# B&R Automation Studio project Tmp_Recorder_V1
Automation Studio 4.5.5.113 SP; technology packages: mapp 5.8.1, mappView 5.8.1

## Configuration X20CPU

CPU X20CP1583, AutomationRuntime B4.53, Build 4.1.2, Vc V4.52.0

CPU X20CP3687X, AutomationRuntime C4.90, Build 4.1.2, Vc V4.52.0

### Task classes (Cpu.sw)
```
Cyclic#8:
  Recorder_1 <- mappRecorder.Recorder_1.prg
Binaries: udbdef, mvLoader, TCData, arsvcreg, Config, sysconf, ashwd, ashwac, asfw, iomap, Role, User, arconfig, OpcUaMap
Libraries: FileIO, runtime, AsBrStr, standard, AsBrWStr, MpBase, sys_lib, IecCheck, asieccon, AsIODiag, MpData, DataObj, brsystem, astime, MpServer, MpFile, AsHttp, AsMem
```

### Task classes (Cpu.sw)
```
Cyclic#4:
  YourTask <- mappRecorder.YourTask.prg
Cyclic#8:
  Recorder_1 <- mappRecorder.Recorder_1.prg
Binaries: udbdef, mvLoader, TCData, arsvcreg, Config, sysconf, ashwd, ashwac, asfw, iomap, Role, User, arconfig, OpcUaMap
Libraries: FileIO, runtime, AsBrStr, standard, AsBrWStr, MpBase, sys_lib, IecCheck, asieccon, AsIODiag, MpData, DataObj, brsystem, astime, MpServer, MpFile, AsHttp, AsMem, MpCom
```

### Hardware
```
X20CP3687X : X20CP3687X v1.7.2.0
  Connector IF2:
    ActivateDevice = 1
  Connector IF3:
    DNAConfiguration = manual
    CycleTime = 2000
  ConfigurationID = Tmp_Recorder
  UserPartitionSize = 200
  AutomaticTransferOfUserfiles = on
  VolatileGlobalPvSize = 300000
  Cyclic8Stack = 20000
  FileDevice1
  FileDeviceName1 = RECORDER_DEVICE
  FileDevicePath1 = F:/
  FileDevice2
  FileDeviceName2 = SIM_DEVICE
  FileDevicePath2 = C:/Temp
  FtpUser1
  FtpUsername1 = br
  FtpUserPassword1 = B+jJgvp9Np1Nx73dPwFagqyDiJQWzomgOnJThoU8F9Q=  // password
  FtpUserSalt1 = Snq9ellj
  FTPAccessRight1 = 0
  ActivateSdm = 0
  ActivateOpcUa = 1
  OpcUaInformationModels_PV_Version = 1
```

### Config_1.mpdatarecorder - X20CP1583/mappServices/Config_1.mpdatarecorder
```
Element gDataRecorder_1 (Type=mpdatarecorder)
```

- Physical/X20CPU/X20CP3687X/mappServices/Config_1.mpdatarecorder: same as Physical/X20CPU/X20CP1583/mappServices/Config_1.mpdatarecorder
## Logical view

Binary libraries used (declarations not repeated): operator, runtime, astime, AsIecCon, FileIO, AsBrStr, AsBrWStr, standard, sys_lib, IecCheck, AsIODiag, DataObj, brsystem, AsHttp, AsMem, MpFile 5.15.0, MpBase 5.15.0, MpCom 5.15.0, MpData 5.15.0, MpServer 5.15.0

### Package Logical/Libraries - Global libraries

- Visualisation Logical/mappView (not shown)

### DatTypes.typ
```iecst
(*------------------------------------------------------------------------------------------------------------------------------------------------------------------------------------------------------------------------*)
(*Global enumerations*)

TYPE
	datSTATE :
		( (*Recorder managment state machine*)
		DAT_WAIT,
		DAT_REG_VAR,
		DAT_READ_DIR,
		DAT_READ_DIR_1,
		DAT_READ_DIR_2,
		DAT_READ_DIR_3,
		DAT_CFG_READ,
		DAT_CFG_WRITE,
		DAT_RECORD,
		DAT_DELETE,
		DAT_VIEW,
		DAT_DOWNLOAD,
		DAT_DOWNLOAD_1,
		DAT_DOWNLOAD_2,
		DAT_DOWNLOAD_3,
		DAT_DOWNLOAD_4,
		DAT_LOAD_VARS,
		DAT_LOAD_VARS_1,
		DAT_LOAD_VARS_2,
		DAT_LOAD_VARS_3,
		DAT_ERROR
		);
END_TYPE

(*------------------------------------------------------------------------------------------------------------------------------------------------------------------------------------------------------------------------*)
(*Global structure*)

TYPE
	datERR : 	STRUCT  (*Recorder managment error structure*)
		Text : WSTRING[200]; (* Error text *)
		State : datSTATE; (* Error step *)
	END_STRUCT;
	datCMD : 	STRUCT  (*Recorder managment command structure*)
		Init : BOOL := TRUE; (*Initialize recorder structure*)
		Record : BOOL; (*Enable recording*)
		Trigger : BOOL; (*Trigger recording*)
		Delete : BOOL; (*Delete selected file *)
		View : BOOL; (*View selected file*)
		Download : BOOL; (*Download selected file*)
		LoadConfig : BOOL; (*Load variable configuration from file*)
		ErrorReset : BOOL; (*Reset pending errors*)
	END_STRUCT;
	datPAR : 	STRUCT  (*Recorder managment parameter structure*)
		RecordName : STRING[DAT_NAME_LENGTH]; (*Record name for command delete and view*)
		RecordNameNew : STRING[DAT_NAME_LENGTH]; (*Record name for command record*)
		RecordMode : MpDataRecordModeEnum; (*Recording mode*)
		RecordInterval : TIME := T#2000ms;
		IsRecording : BOOL; (*Indicates that recording is active*)
		SamplesNum : UDINT; (*Number of recorded samples*)
		Initialized : BOOL; (*Indicates that recorder managment was initialized*)
		VisuSlotID : USINT; (*ID for connected web connection*)
	END_STRUCT;
	datDAT : 	STRUCT  (*Recorder managment data structure*)
		RecordNames : ARRAY[0..DAT_MAX_NUM]OF STRING[DAT_NAME_LENGTH]; (*Recorder unicode name*)
		RecordNum : UINT; (*Number of recorded files*)
	END_STRUCT;
	datVIS : 	STRUCT  (*Recorder managment visualization structure*)
		RecordNames : ARRAY[0..DAT_MAX_NUM]OF STRING[DAT_VIS_LENGTH]; (*Recorder file size*)
		RecordNum : UINT; (*Number of records*)
		RecordFilter : STRING[DAT_NAME_LENGTH]; (*Filter for record names*)
		RecordSelected : STRING[DAT_VIS_LENGTH]; (*Selected record for command delete or view*)
		RecordDoubleClick : USINT; (*TrackDoubleClick event*)
		EnableButtons : BOOL;
		ViewFilePath : STRING[DAT_VIS_LENGTH]; (*Full path for viewing file*)
		ViewFile : BOOL; (*Show message box on error*)
		DownloadFileUrl : STRING[200]; (*File upload and download url*)
		ShowMessageBoxError : BOOL; (*Show message box on error*)
	END_STRUCT;
	datMAIN : 	STRUCT  (*Recorder managment main structure*)
		CMD : datCMD; (*Command structure *)
		PAR : datPAR; (*Parameter structure *)
		DAT : datDAT; (*Data structure*)
		VIS : ARRAY[0..DAT_MAX_CLIENTS_ID]OF datVIS; (*Visualization structure*)
		ERR : datERR; (*Error structure *)
		StatusText : WSTRING[100]; (*Shows the result of the last command*)
		StatusNo : DINT; (*Error number *)
	END_STRUCT;
END_TYPE

(*------------------------------------------------------------------------------------------------------------------------------------------------------------------------------------------------------------------------*)
(*Structure that contains the recorder variables*)

TYPE
	datVariable : 	STRUCT
		Temperature1 : INT := 11;
		Temperature2 : INT := 22;
		MotorSpeed : DINT := 33;
		Position : REAL := 44.55;
	END_STRUCT;
END_TYPE
```

### DatVariables.var
```iecst
(*------------------------------------------------------------------------------------------------------------------------------------------------------------------------------------------------------------------------*)
(*Configuration for recorder managment*)
VAR CONSTANT
	DAT_MAX_NUM : USINT := 100; (*Maximum number of record files*)
	DAT_NAME_LENGTH : USINT := 40; (*Maximum length for a record name*)
	DAT_VIS_LENGTH : USINT := 120; (*Make this DAT_NAME_LENGTH  x3*)
	DAT_MAX_CLIENTS_ID : USINT := 2; (*Highest client ID for concurrent web client connections. Do not change this number.*)
END_VAR
VAR
	DAT_VIEW_FILTER : ARRAY[0..9] OF STRING[5] := ['csv','pdf',8('')]; (*Files extensions than can be used with the view command*)
END_VAR
VAR CONSTANT
	DAT_DOWNLOAD_SIZE : UDINT := 500000; (*Maximum size of memory allocated for uploading and downloading files*)
	DAT_VAR_NUM : USINT := 10; (*Maximum number of variables that can be registered*)
	DAT_THIS_TASK : STRING[40] := 'Recorder_1'; (*Name of this task and the global variables structure*)
	DAT_DEVICE : STRING[80] := 'RECORDER_DEVICE'; (*Device name for the recorder data defined under File Devices in the CPU configuration*)
	DAT_CONFIG : STRING[80] := 'var_list.csv'; (*File with a list of variables in CSV format*)
END_VAR
VAR
	DAT_MPLINK : {REDUND_UNREPLICABLE} STRING[80] := 'gDataRecorder_1'; (*mappRecoreer link name from configuration view*)
END_VAR
(*------------------------------------------------------------------------------------------------------------------------------------------------------------------------------------------------------------------------*)
(*Add you variables to this list*)
VAR
	DAT_VAR_LIST : ARRAY[1..DAT_VAR_NUM] OF STRING[100] := ['YourTask:Temperature1','YourTask:Temperature2','YourTask:MotorSpeed','YourTask:Position',6('')]; (*List of variables to be inlcuded in a record*)
	Recorder_1 : datMAIN; (*Global record structure. The name must match the task name of the recorder managment.*)
END_VAR
```

### Program Logical/mappRecorder/Recorder_1 (IEC)

#### Init.st - Init and local configuration
```iecst
// -------------------------------------------------------------------------------------------------------------------
//	Function:	Data recorder management with mappData
// -------------------------------------------------------------------------------------------------------------------
PROGRAM _INIT
	// ----------------------------------------------------------------------------------------
	// The following settings can be adjusted
	IF(DiagCpuIsSimulated()) THEN
		DeviceName 	:= 'SIM_DEVICE';	// Device name from the CPU configuration for simulation
	ELSE
		DeviceName 	:= DAT_DEVICE;		// Device name from the CPU configuration for X20CPU
	END_IF

	// ----------------------------------------------------------------------------------------
	// Dont change anything below this line
	// ----------------------------------------------------------------------------------------

	// ----------------------------------------------------------------------------------------
	// Make sure global variable structure and task name are correct
	taskStatus := ST_ident(ADR(DAT_THIS_TASK), taskGroup, ADR(taskID));
	pvStatus := PV_xgetadr(ADR(DAT_THIS_TASK), ADR(pvADR), ADR(pvLEN));
	// Connect global and local structure
	IF(pvStatus = 0) THEN
		RECORDER ACCESS pvADR;
		brsmemset(ADR(RECORDER.ERR), 0 , SIZEOF(RECORDER.ERR));
		RECORDER.PAR.Initialized := FALSE;
	END_IF

	// ----------------------------------------------------------------------------------------
	// Get mapp link information
	MpComGetLink_0.Enable := TRUE;
	MpComGetLink_0.ComponentName := ADR(DAT_MPLINK);
	MpComGetLink_0();
	// Create error
	IF(MpComGetLink_0.Error) THEN
		rec_state := CreateError(ADR(RECORDER), ERR_DAT_MPLINK, "mplink name is incorrect", rec_state);
	END_IF

	// ----------------------------------------------------------------------------------------
	// Allocate memory for file upload and download
	AsMemPartCreate_0.enable	:= TRUE;
	AsMemPartCreate_0.len		:= DAT_DOWNLOAD_SIZE;
	AsMemPartCreate_0();
	IF AsMemPartCreate_0.status <> 0 THEN
		CreateError(ADR(RECORDER), ERR_MEM_ALLOC, "file upload and download alloc failed", rec_state);
	ELSE
		AsMemPartAllocClear_0.enable	:= TRUE;
		AsMemPartAllocClear_0.ident		:= AsMemPartCreate_0.ident;
		AsMemPartAllocClear_0.len		:= DAT_DOWNLOAD_SIZE;
		AsMemPartAllocClear_0();
		IF AsMemPartCreate_0.status <> 0 THEN
			CreateError(ADR(RECORDER), ERR_MEM_ALLOC, "file upload and download clear failed", rec_state);
		END_IF
	END_IF
END_PROGRAM
```

#### Main.st - Cyclic code
```iecst
// -------------------------------------------------------------------------------------------------------------------
//	Cylic task for data recorder management
// -------------------------------------------------------------------------------------------------------------------
PROGRAM _CYCLIC
	// --------------------------------------------------------------------------------------------------------------------
	// Make sure task name and global structure correct
	IF(pvStatus <> 0) THEN
		RETURN;
	END_IF
	IF(taskStatus <> 0) THEN
		rec_state := CreateError(ADR(RECORDER), ERR_DAT_TASK_NAME, "Task name is incorrect", rec_state);
		RETURN;
	END_IF

	// --------------------------------------------------------------------------------------------------------------------
	// Make sure we dont exceed maximum number of web clients
	IF(RECORDER.PAR.VisuSlotID > DAT_MAX_CLIENTS_ID) THEN
		rec_state := CreateError(ADR(RECORDER), ERR_DAT_TOO_MANY_CLIENTS, "More than 3 clients try to connect to data recorder", rec_state);
		RETURN;
	END_IF

	// --------------------------------------------------------------------------------------------------------------------
	// Cyclic function calls
	MpDataRecorder_0();
	RECORDER.PAR.IsRecording := MpDataRecorder_0.Recording;
	RECORDER.PAR.SamplesNum := MpDataRecorder_0.Info.TotalSamples;
	MpDataRecorder_0.RecordMode := RECORDER.PAR.RecordMode;
	MpDataRecorder_0.SamplingTime := RECORDER.PAR.RecordInterval;

		// -------------------------------------------------------------------------------------------------------------------
	// Recorder managment state machine
		// -------------------------------------------------------------------------------------------------------------------
	CASE rec_state OF
		// --------------------------------------------------------------------------------------------------------------------
		// Wait for command
		// --------------------------------------------------------------------------------------------------------------------
		DAT_WAIT:
			// Set OK state
			RECORDER.StatusNo := ERR_OK;
			// --------------------------------------------------------------------------------------------------------------------
			// Track filter change and data refresh
			IF ((brwcscmp(ADR(RecordFilterOld[VisuSlotID]), ADR(RECORDER.VIS[VisuSlotID].RecordFilter)) <> 0) OR (RecordNumOld[VisuSlotID] <> RECORDER.DAT.RecordNum)) THEN
				brsmemset(ADR(RECORDER.VIS[VisuSlotID].RecordNames), 0, SIZEOF(RECORDER.VIS[VisuSlotID].RecordNames));
				idy := 0;
				IF(RECORDER.DAT.RecordNum > 0) THEN
					FOR idx:=0 TO RECORDER.DAT.RecordNum - 1 DO
						// --------------------------------------------------------------------------------
						// Verify that file name contains filter
						IF (brsstrlen(ADR(RECORDER.VIS[VisuSlotID].RecordFilter)) = 0 OR IsInstr(ADR(RECORDER.DAT.RecordNames[idx]), ADR(RECORDER.VIS[VisuSlotID].RecordFilter))) > 0 THEN
							String2DataProvider(ADR(RECORDER.DAT.RecordNames[idx]), ADR(tmpStr1));
							RECORDER.VIS[VisuSlotID].RecordNames[idy] := tmpStr1;
							idy := idy + 1;
						END_IF
					END_FOR;
					brsstrcpy(ADR(RecordFilterOld[VisuSlotID]), ADR(RECORDER.VIS[VisuSlotID].RecordFilter));
				END_IF
				RecordNumOld[VisuSlotID] := RECORDER.DAT.RecordNum;
				RECORDER.VIS[VisuSlotID].RecordNum := idy;
				// Enable/Disable delete button
				IF(RECORDER.VIS[VisuSlotID].RecordNum > 0) THEN
					RECORDER.VIS[VisuSlotID].EnableButtons := TRUE;
				ELSE
					RECORDER.VIS[VisuSlotID].EnableButtons := FALSE;
				END_IF
			END_IF

			// ------------------------------------------------------------------------------------------------
			// Handle double click for file open
			IF(RECORDER.VIS[VisuSlotID].RecordDoubleClick > 0) THEN
				DoubleClickRecordName[VisuSlotID].PT := 50;
				DoubleClickRecordName[VisuSlotID].IN := 1;
				DoubleClickRecordName[VisuSlotID]();
				// Open selected file
				IF(RECORDER.VIS[VisuSlotID].RecordDoubleClick > 1) THEN
					DoubleClickRecordName[VisuSlotID].IN := 0;
					DoubleClickRecordName[VisuSlotID]();
					RECORDER.VIS[VisuSlotID].RecordDoubleClick := 0;
					RECORDER.PAR.VisuSlotID := VisuSlotID;
					RECORDER.CMD.View := TRUE;
				END_IF
			END_IF
			IF(DoubleClickRecordName[VisuSlotID].Q) THEN
				DoubleClickRecordName[VisuSlotID].IN := 0;
				DoubleClickRecordName[VisuSlotID]();
				IF(RECORDER.VIS[VisuSlotID].RecordDoubleClick > 0) THEN
					RECORDER.VIS[VisuSlotID].RecordDoubleClick := RECORDER.VIS[VisuSlotID].RecordDoubleClick - 1;
				END_IF
			END_IF

			// Cylce through the client web seesions
			VisuSlotID := VisuSlotID + 1;
			IF(VisuSlotID > DAT_MAX_CLIENTS_ID) THEN
				VisuSlotID := 0;
			END_IF

			// ----------------------------------------------------------------------------------------
			// Command refresh
			IF (RECORDER.CMD.Init = TRUE) THEN
				// Reset data structure and trigger name refresh for vis
				brsmemset(ADR(RECORDER.DAT), 0, SIZEOF(RECORDER.DAT));
				brsmemset(ADR(RecordNumOld), 16#FF, SIZEOF(RecordNumOld));
				pvCnt := 1;
				rec_state := DAT_CFG_READ;
			// ----------------------------------------------------------------------------------------
			// Command continues recording
			ELSIF (RECORDER.CMD.Record = TRUE) THEN
				tmpWStr1 := "continues recording...";
				rec_state := DAT_CFG_WRITE;
			// ----------------------------------------------------------------------------------------
			// Command trigger recording
			ELSIF (RECORDER.CMD.Trigger = TRUE) THEN
				tmpWStr1 := "recording by trigger...";
				rec_state := DAT_RECORD;
			// ----------------------------------------------------------------------------------------
			// Command delete recording
			ELSIF (RECORDER.CMD.Delete = TRUE AND RECORDER.PAR.RecordName <> '') THEN
				animation := WorkingStatus(ADR(RECORDER), ADR("deleting recording..."), animation);
				RecordName := RECORDER.PAR.RecordName;
				rec_state := DAT_DELETE;
			// ----------------------------------------------------------------------------------------
			// Command view file
			ELSIF (RECORDER.CMD.View = TRUE AND RECORDER.VIS[RECORDER.PAR.VisuSlotID].RecordSelected <> '') THEN
				RECORDER.VIS[RECORDER.PAR.VisuSlotID].ViewFilePath := '';
				//RecordName := RECORDER.PAR.RecordName;
				rec_state := DAT_VIEW;
			// ----------------------------------------------------------------------------------------
			// Download selected file
			ELSIF (RECORDER.CMD.Download = 1 AND RECORDER.PAR.RecordName <> '') THEN
				RECORDER.VIS[RECORDER.PAR.VisuSlotID].DownloadFileUrl := '';
				RecordName := RECORDER.PAR.RecordName;
				rec_state := DAT_DOWNLOAD;
			// ----------------------------------------------------------------------------------------
			// Load variable configuration file
			ELSIF (RECORDER.CMD.LoadConfig = 1) THEN
				rec_state := DAT_LOAD_VARS;
			END_IF

			// ----------------------------------------------------------------------------------------
			// Check parameters
			IF (RECORDER.CMD.Init OR RECORDER.CMD.Delete OR RECORDER.CMD.View OR RECORDER.CMD.Download OR RECORDER.CMD.LoadConfig OR RECORDER.CMD.Record) THEN
				// Set busy state
				RECORDER.StatusNo := ERR_FUB_BUSY;
				// Make sure recorder was intialized
				IF (NOT RECORDER.CMD.Init AND (RECORDER.CMD.Delete OR RECORDER.CMD.View) AND NOT RECORDER.PAR.Initialized) THEN
					rec_state := CreateError(ADR(RECORDER), ERR_DAT_NOT_INITIALIZED, "recorder is not initialized", rec_state);
				END_IF
				// Make sure device name is valid
				IF(DeviceName = '') THEN
					rec_state := CreateError(ADR(RECORDER), ERR_DAT_DEV_NAME_EMPTY, "device name is empty", rec_state);
				END_IF
				// Make sure record name is valid
				IF(RECORDER.PAR.RecordName = '' AND (RECORDER.CMD.Delete OR RECORDER.CMD.Download)) THEN
					rec_state := CreateError(ADR(RECORDER), ERR_DAT_NAME_EMPTY, "record name is empty", rec_state);
				END_IF
				// Make sure record name is valid
				IF(RECORDER.PAR.RecordNameNew = '' AND RECORDER.CMD.Record) THEN
					rec_state := CreateError(ADR(RECORDER), ERR_DAT_NAME_EMPTY, "new record name is empty", rec_state);
				END_IF
				// Make sure variable name has at least one entry
				IF(DAT_VAR_LIST[1] = '' AND NOT RECORDER.CMD.LoadConfig) THEN
					rec_state := CreateError(ADR(RECORDER), ERR_DAT_VAR_NAME_EMPTY, "variable name is empty", rec_state);
				END_IF
			END_IF

		// ----------------------------------------------------------------------------------------------------------------------------------
		// Read data configuration
		// ----------------------------------------------------------------------------------------------------------------------------------
		DAT_CFG_READ:
			// Read data configuration
			mappDataCfg.Load := TRUE;

			// ----------------------------------------------------------------------------------------------------------------------------------
			// OK
			IF (mappDataCfg.CommandDone AND NOT mappDataCfg.Error) THEN
				// Reset config function block
				mappDataCfg.Load := FALSE;
				RECORDER.PAR.RecordNameNew := MpDataRecorderCfg.FileNamePattern;
				rec_state := DAT_REG_VAR;
				// ----------------------------------------------------------------------------------------------------------------------------------
				// Error
			ELSIF(mappDataCfg.Error) THEN
				rec_state := CreateError(ADR(RECORDER), mappDataCfg.StatusID, "error reading configuration", rec_state);
			END_IF

		// --------------------------------------------------------------------------------------------------------------------
		// Register variable structure
		// --------------------------------------------------------------------------------------------------------------------
		DAT_REG_VAR:
			MpRecorderRegPar_0[pvCnt].Enable := 1;
			MpRecorderRegPar_0[pvCnt].MpLink := ADR(MpComGetLink_0.MpLink);
			MpRecorderRegPar_0[pvCnt].PVName := ADR(DAT_VAR_LIST[pvCnt]);

			// ----------------------------------------------------------------------------------------
			// OK
			IF (MpRecorderRegPar_0[pvCnt].Active AND NOT MpRecorderRegPar_0[pvCnt].Error) THEN
				pvCnt := pvCnt + 1;
				// Register next variable
				IF((pvCnt >= SIZEOF(DAT_VAR_LIST)/SIZEOF(DAT_VAR_LIST[pvCnt])) OR (DAT_VAR_LIST[pvCnt] = '')) THEN
					rec_state := DAT_READ_DIR;
				END_IF
			// ----------------------------------------------------------------------------------------
			// Error
			ELSIF (MpRecorderRegPar_0[pvCnt].Error) THEN
				tmpWStr1 := "error trying to register variable name ";
				brwcsconv(ADR(tmpWStr2), ADR(DAT_VAR_LIST[pvCnt]), brwU8toUC);
				brwcscat(ADR(tmpWStr1), ADR(tmpWStr2));
				rec_state := CreateError(ADR(RECORDER), MpRecorderRegPar_0[pvCnt].StatusID, tmpWStr1, rec_state);
			END_IF
		// --------------------------------------------------------------------------------------------------------------------
		// Read directory information
		// --------------------------------------------------------------------------------------------------------------------
		DAT_READ_DIR:
			// Show current state
			animation := WorkingStatus(ADR(RECORDER), ADR("reading records..."), animation);
			// ----------------------------------------------------------------------------------------
			// Clear all entrys
			brsmemset(ADR(RECORDER.DAT), 0, SIZEOF(RECORDER.DAT));
			RECORDER.DAT.RecordNum := 0;
			// ----------------------------------------------------------------------------------------
			// Set values and get device dir
			DInfo.enable 	:= 1;
			DInfo.pDevice	:= ADR(DeviceName);
			DInfo();

			// ----------------------------------------------------------------------------------------
			// OK
			IF (DInfo.status = OK) THEN
				rec_state := DAT_READ_DIR_1;
			ELSIF (DInfo.status = fiERR_DEVICE_MANAGER) THEN
				tmpWStr1 := "file device ";
				brwcsconv(ADR(tmpWStr2), ADR(DeviceName), brwU8toUC);
				brwcscat(ADR(tmpWStr1), ADR(tmpWStr2));
				brwcscat(ADR(tmpWStr1), ADR(" is unavailable"));
				rec_state := CreateError(ADR(RECORDER), DInfo.status, tmpWStr1, rec_state);
			// ----------------------------------------------------------------------------------------
			// Error
			ELSIF (DInfo.status <> ERR_FUB_BUSY) THEN
				rec_state := CreateError(ADR(RECORDER), DInfo.status, "error dir info", rec_state);
			END_IF
		// --------------------------------------------------------------------------------------------------------------------
		// Open directory
		// --------------------------------------------------------------------------------------------------------------------
		DAT_READ_DIR_1:
			DOpen.enable 	:= 1;
			DOpen.pDevice	:= ADR(DeviceName);
			DOpen();

			// ----------------------------------------------------------------------------------------
			// OK
			IF (DOpen.status = OK) THEN
				has_oversized_items := FALSE;
				rec_state := DAT_READ_DIR_2;
			// ----------------------------------------------------------------------------------------
			// Error
			ELSIF (DOpen.status <> ERR_FUB_BUSY) THEN
				rec_state := CreateError(ADR(RECORDER), DOpen.status, "error dir open", rec_state);
			END_IF;
		// --------------------------------------------------------------------------------------------------------------------
		// Read file directory information
		// --------------------------------------------------------------------------------------------------------------------
		DAT_READ_DIR_2:
			DRead.enable 	:= 1;
			DRead.ident		:= DOpen.ident;
			DRead.pData 	:= ADR(lDirReadData);
			DRead.data_len 	:= SIZEOF(lDirReadData);
			DRead();

			// ----------------------------------------------------------------------------------------
			// OK
			IF (DRead.status = OK AND lDirReadData.Mode = fiFILE) THEN
				animation := WorkingStatus(ADR(RECORDER), ADR("reading record data..."), animation);
				// Make sure file name does not exceed maximum string size
				IF (brsstrlen(ADR(lDirReadData.Filename)) < DAT_NAME_LENGTH) THEN
					// Copy dir info to string
					brsmemset(ADR(RECORDER.PAR.RecordName), 0, SIZEOF(RECORDER.PAR.RecordName));
					brsstrcpy(ADR(RECORDER.PAR.RecordName), ADR(lDirReadData.Filename));
					// Make sure file extension is CSV or PDF
					IF(brsstrlen(ADR(RECORDER.PAR.RecordName)) > 4 AND ((brsmemcmp(ADR(RECORDER.PAR.RecordName) + (brsstrlen(ADR(RECORDER.PAR.RecordName)) - 4), ADR('.csv'), 4) = 0) OR (brsmemcmp(ADR(RECORDER.PAR.RecordName) + (brsstrlen(ADR(RECORDER.PAR.RecordName)) - 4), ADR('.pdf'), 4) = 0))) THEN
						// ------------------------------------------------------------------------------------
						// Verify that we still have space in list
						IF (RECORDER.DAT.RecordNum <= DAT_MAX_NUM) THEN
							// Generate ASCII data, insert record into list
							InsertRecName(ADR(RECORDER), RECORDER.PAR.RecordName);
							// Error
						ELSE
							rec_state := CreateError(ADR(RECORDER), ERR_DAT_MAX_NUM, "maximum number of records reached", rec_state);
						END_IF
					END_IF
				ELSE
					has_oversized_items := TRUE;
				END_IF
			// ----------------------------------------------------------------------------------------
			// Last entry reached
			ELSIF (DRead.status = fiERR_NO_MORE_ENTRIES) THEN
				rec_state := DAT_READ_DIR_3;
			// ----------------------------------------------------------------------------------------
			// Error
			ELSIF (DRead.status <> ERR_FUB_BUSY AND DRead.status <> OK) THEN
				rec_state := CreateError(ADR(RECORDER), DRead.status, "error record list read", rec_state);
			END_IF
		// --------------------------------------------------------------------------------------------------------------------
		// Close directory information
		// --------------------------------------------------------------------------------------------------------------------
		DAT_READ_DIR_3:
			DClose.enable 	:= 1;
			DClose.ident	:= DOpen.ident;
			DClose();

			// ----------------------------------------------------------------------------------------
			// OK
			IF (DClose.status = OK) THEN
				// Reset command and return to wait state
				RECORDER.StatusText	:= "initializing complete";
				RECORDER.CMD.Init := 0;
				RECORDER.CMD.LoadConfig := 0;
				RECORDER.CMD.Delete := 0;
				RECORDER.PAR.Initialized := TRUE;
				DClose.ident := 0;
				IF(has_oversized_items) THEN
					rec_state := CreateError(ADR(RECORDER), ERR_DAT_NAME_LENGTH, "one or more record names exceeds maximum length", rec_state);
				ELSE
					rec_state := DAT_WAIT;
				END_IF
			// ----------------------------------------------------------------------------------------
			// Error
			ELSIF (DClose.status <> ERR_FUB_BUSY) THEN
				rec_state := CreateError(ADR(RECORDER), DClose.status, "error dir close", rec_state);
			END_IF

		// ----------------------------------------------------------------------------------------------------------------------------------
		// Write data configuration
		// ----------------------------------------------------------------------------------------------------------------------------------
		DAT_CFG_WRITE:
			// Make sure file extension is CSV or PDF
			IF(brsstrlen(ADR(RECORDER.PAR.RecordNameNew)) <= 4 OR ((brsmemcmp(ADR(RECORDER.PAR.RecordNameNew) + (brsstrlen(ADR(RECORDER.PAR.RecordNameNew)) - 4), ADR('.csv'), 4) <> 0) AND (brsmemcmp(ADR(RECORDER.PAR.RecordNameNew) + (brsstrlen(ADR(RECORDER.PAR.RecordNameNew)) - 4), ADR('.pdf'), 4) <> 0))) THEN
				// Make sure record name is not too large with extension
				IF(brsstrlen(ADR(RECORDER.PAR.RecordNameNew)) <= SIZEOF(RECORDER.PAR.RecordNameNew) - 4) THEN
					IF(MpDataRecorderCfg.Format.FileType = mpDATA_FILE_TYPE_CSV) THEN
						brsstrcat(ADR(RECORDER.PAR.RecordNameNew), ADR('.csv'));
					ELSE
						brsstrcat(ADR(RECORDER.PAR.RecordNameNew), ADR('.pdf'));
					END_IF
				ELSE
					rec_state := CreateError(ADR(RECORDER), ERR_DAT_NAME_LENGTH, "record name exceeds maximum size", rec_state);
					RETURN;
				END_IF
			END_IF

			// Write data configuration
			mappDataCfg.Enable := TRUE;
			mappDataCfg.MpLink := ADR(MpComGetLink_0.MpLink);
			MpDataRecorderCfg.FileNamePattern := RECORDER.PAR.RecordNameNew;
			mappDataCfg.Configuration := ADR(MpDataRecorderCfg);
			mappDataCfg.Save := TRUE;

			// ----------------------------------------------------------------------------------------------------------------------------------
			// OK
			IF (mappDataCfg.CommandDone AND NOT mappDataCfg.Error) THEN
				// Reset config function block
				mappDataCfg.Save := FALSE;
				rec_state := DAT_RECORD;
			// ----------------------------------------------------------------------------------------------------------------------------------
			// Error
			ELSIF(mappDataCfg.Error) THEN
				rec_state := CreateError(ADR(RECORDER), mappDataCfg.StatusID, "error writing configuration", rec_state);
			END_IF

		// --------------------------------------------------------------------------------------------------------------------
		// Record data
		// --------------------------------------------------------------------------------------------------------------------
		DAT_RECORD:
			// Set busy state
			RECORDER.StatusNo := ERR_FUB_BUSY;
			animation := WorkingStatus(ADR(RECORDER), ADR(tmpWStr1), animation);

			IF (MpDataRecorder_0.Active) THEN
				MpDataRecorder_0.Record := RECORDER.CMD.Record OR RECORDER.CMD.Trigger;
			END_IF;

			// ----------------------------------------------------------------------------------------
			// OK
			IF (MpDataRecorder_0.Recording AND NOT MpDataRecorder_0.Error AND MpDataRecorder_0.StatusID = 0) THEN
				// Command record by trigger
				IF(RECORDER.CMD.Trigger) THEN
					// Fire trigger when recording is engaged
					IF (NOT MpDataRecorder_0.Trigger) THEN
						MpDataRecorder_0.Trigger := TRUE;
						// Reset trigger when event was recorded
					ELSE
						MpDataRecorder_0.Trigger := FALSE;
						RECORDER.CMD.Trigger := FALSE;
						IF(NOT RECORDER.CMD.Record) THEN
							MpDataRecorder_0.Record := FALSE;
							RECORDER.StatusText := "created new record by trigger";
							rec_state := DAT_READ_DIR;
						END_IF
					END_IF
				// Recording disabled
				ELSIF (NOT RECORDER.CMD.Record) THEN
					rec_state := DAT_READ_DIR;
				END_IF
			// ----------------------------------------------------------------------------------------
			// Error
			ELSIF (MpDataRecorder_0.Error OR MpDataRecorder_0.StatusID <> 0) THEN
				rec_state := CreateError(ADR(RECORDER), MpDataRecorder_0.StatusID, "error trying to create record", rec_state);
			END_IF
		// --------------------------------------------------------------------------------------------------------------------
		// Delete selected record
		// --------------------------------------------------------------------------------------------------------------------
		DAT_DELETE:
			// ----------------------------------------------------------------------------------------
			// Initialize file delete structure
			FDelete.enable		:= 1;
			FDelete.pDevice 	:= ADR(DeviceName);
			FDelete.pName		:= ADR(RecordName);
			FDelete();

			// ----------------------------------------------------------------------------------------
			// OK
			IF (FDelete.status = OK) THEN
				CreateMessage(ADR(RECORDER.StatusText), ADR("deleted record"), ADR(RECORDER.PAR.RecordName), RECORDER.PAR.VisuSlotID);
				rec_state := DAT_READ_DIR;
			// ----------------------------------------------------------------------------------------
			// Error
			ELSIF (FDelete.status <> ERR_FUB_BUSY) THEN
				tmpWStr1 := "error deleting record ";
				brwcsconv(ADR(tmpWStr2), ADR(RecordName), brwU8toUC);
				brwcscat(ADR(tmpWStr1), ADR(tmpWStr2));
				rec_state := CreateError(ADR(RECORDER), FDelete.status, tmpWStr1, rec_state);
			END_IF
		// --------------------------------------------------------------------------------------------------------------------
		// View selected file
		// --------------------------------------------------------------------------------------------------------------------
		DAT_VIEW:
			IF(RECORDER.DAT.RecordNum > 0) THEN
				FOR idx:=0 TO SIZEOF(DAT_VIEW_FILTER)/SIZEOF(DAT_VIEW_FILTER[0]) - 1 DO
					IF(brsstrlen(ADR(RECORDER.VIS[RECORDER.PAR.VisuSlotID].RecordSelected)) >= brsstrlen(ADR(DAT_VIEW_FILTER[idx])) AND DAT_VIEW_FILTER[idx] <> '') THEN
						// --------------------------------------------------------------------------------
						// Verify that file name contains filter
						IF(brsmemcmp(ADR(RECORDER.VIS[RECORDER.PAR.VisuSlotID].RecordSelected) + brsstrlen(ADR(RECORDER.VIS[RECORDER.PAR.VisuSlotID].RecordSelected)) - brsstrlen(ADR(DAT_VIEW_FILTER[idx])) , ADR(DAT_VIEW_FILTER[idx]), brsstrlen(ADR(DAT_VIEW_FILTER[idx]))) = 0) THEN
							RECORDER.VIS[RECORDER.PAR.VisuSlotID].ViewFilePath := '/FileDevice:';
							brsstrcat(ADR(RECORDER.VIS[RECORDER.PAR.VisuSlotID].ViewFilePath), ADR(DeviceName));
							brsstrcat(ADR(RECORDER.VIS[RECORDER.PAR.VisuSlotID].ViewFilePath), ADR("/"));
							brsstrcat(ADR(RECORDER.VIS[RECORDER.PAR.VisuSlotID].ViewFilePath), ADR(RECORDER.VIS[RECORDER.PAR.VisuSlotID].RecordSelected));
							RECORDER.CMD.View := FALSE;
							RECORDER.VIS[RECORDER.PAR.VisuSlotID].ViewFile := TRUE;
							rec_state := DAT_WAIT;
							RETURN;
						END_IF
					END_IF
				END_FOR;
				RECORDER.StatusText := "error this file extension is not supported for viewing";
				RECORDER.CMD.View := FALSE;
				rec_state := DAT_WAIT;
			END_IF
		// --------------------------------------------------------------------------------------------------------------------
		// Download file
		// --------------------------------------------------------------------------------------------------------------------
		DAT_DOWNLOAD:
			// ----------------------------------------------------------------------------------------
			// Initialize file open structure
			FOpen.enable	:= TRUE;
			FOpen.pDevice 	:= ADR(DeviceName);
			FOpen.pFile		:= ADR(RecordName);
			FOpen();

			// ----------------------------------------------------------------------------------------
			// OK
			IF (FOpen.status = OK) THEN
				// Make sure file fits into memory
				IF(FOpen.filelen <= DAT_DOWNLOAD_SIZE) THEN
					// Clear memory and reset web service
					brsmemset(AsMemPartAllocClear_0.mem, 0, DAT_DOWNLOAD_SIZE);
					WebserviceDownload.enable := FALSE;
					WebserviceDownload();
					rec_state := DAT_DOWNLOAD_1;
					// File is too large
				ELSE
					tmpWStr1 := "download file exceeds maximum buffer size of ";
					brsitoa(DAT_DOWNLOAD_SIZE, ADR(tmpStr1));
					brwcsconv(ADR(tmpWStr2),ADR(tmpStr1), brwU8toUC);
					brwcscat(ADR(tmpWStr1), ADR(tmpWStr2));
					brwcscat(ADR(tmpWStr1), ADR(" bytes"));
					rec_state := CreateError(ADR(RECORDER), ERR_MEM_DOWNLOAD, tmpWStr1, rec_state);
				END_IF;
			// ----------------------------------------------------------------------------------------
			// Error
			ELSIF (FOpen.status <> ERR_FUB_BUSY) THEN
				rec_state := CreateError(ADR(RECORDER), FOpen.status, "error opening file for download", rec_state);
			END_IF
		// --------------------------------------------------------------------------------------------------------------------
		// Download file
		// --------------------------------------------------------------------------------------------------------------------
		DAT_DOWNLOAD_1:
			// ----------------------------------------------------------------------------------------
			// Initialize file read structure
			FRead.enable	:= TRUE;
			FRead.ident		:= FOpen.ident;
			FRead.len		:= FOpen.filelen;
			FRead.pDest		:= AsMemPartAllocClear_0.mem;
			FRead();

			// ----------------------------------------------------------------------------------------
			// OK
			IF (FRead.status = OK) THEN
				rec_state := DAT_DOWNLOAD_2;
			// ----------------------------------------------------------------------------------------
			// Error
			ELSIF (FRead.status <> ERR_FUB_BUSY) THEN
				rec_state := CreateError(ADR(RECORDER), FRead.status, "error reading file for download", rec_state);
			END_IF
		// --------------------------------------------------------------------------------------------------------------------
		// Download file
		// --------------------------------------------------------------------------------------------------------------------
		DAT_DOWNLOAD_2:
			// ----------------------------------------------------------------------------------------
			// Initialize file close structure
			FClose.enable	:= TRUE;
			FClose.ident	:= FOpen.ident;
			FClose();

			// ----------------------------------------------------------------------------------------
			// OK
			IF (FClose.status = OK) THEN
				DownloadTimeout.IN := 0;
				DownloadTimeout();
				rec_state := DAT_DOWNLOAD_3;
			// ----------------------------------------------------------------------------------------
			// Error
			ELSIF (FClose.status <> ERR_FUB_BUSY) THEN
				rec_state := CreateError(ADR(RECORDER), FClose.status, "error closing file for download", rec_state);
			END_IF
		// --------------------------------------------------------------------------------------------------------------------
		// Download file - web service
		// --------------------------------------------------------------------------------------------------------------------
		DAT_DOWNLOAD_3:
			// ----------------------------------------------------------------------------------------
			// Create response header
			ResponseHeaderData :=  'Content-Type: application/octet-stream; Content-Transfer-Encoding: binary; Content-Disposition: attachment; filename="';
			brsstrcpy(ADR(tmpStr1), ADR(RecordName));
			ReplaceString(ADR(tmpStr1), ADR(' '), ADR('%20'), FALSE);
			brsstrcat(ADR(ResponseHeaderData), ADR(tmpStr1));
			brsstrcat(ADR(ResponseHeaderData), ADR('"'));

			// ----------------------------------------------------------------------------------------
			// Pre-configure web service for download
			ResponseHeader.rawHeader.pData 	:= ADR(ResponseHeaderData);
			ResponseHeader.rawHeader.dataSize 	:= SIZEOF(ResponseHeaderData);
			ResponseHeader.rawHeader.dataLen 	:= brsstrlen(ADR(ResponseHeaderData));

			// ----------------------------------------------------------------------------------------
			// Start web service
			WebserviceDownload.enable 			:= TRUE;
			WebserviceDownload.option 			:= httpOPTION_HTTP_10 + httpOPTION_SERVICE_TYPE_NAME;
			WebserviceDownload.pResponseData 	:= AsMemPartAllocClear_0.mem;
			WebserviceDownload.pResponseHeader	:= ADR(ResponseHeader);
			WebserviceDownload.pServiceName 	:= ADR(tmpStr1);
			WebserviceDownload.responseDataLen 	:= FOpen.filelen;
			WebserviceDownload();

			// ----------------------------------------------------------------------------------------
			// Timeout if file is not pulled from browser
			DownloadTimeout.IN := 1;
			DownloadTimeout.PT := 300;
			DownloadTimeout();
			IF(DownloadTimeout.Q) THEN
				rec_state := CreateError(ADR(RECORDER), ERR_TIMEOUT_DOWNLOAD, "error download response timed out", rec_state);
			END_IF

			// ----------------------------------------------------------------------------------------
			// Set URL
			IF (WebserviceDownload.status = ERR_FUB_BUSY AND RECORDER.VIS[RECORDER.PAR.VisuSlotID].DownloadFileUrl = '') THEN
				brsstrcat(ADR(RECORDER.VIS[RECORDER.PAR.VisuSlotID].DownloadFileUrl), ADR(RecordName));
			// Start sending data
			ELSIF (WebserviceDownload.status = OK AND WebserviceDownload.send = FALSE AND RECORDER.VIS[RECORDER.PAR.VisuSlotID].DownloadFileUrl <> '') THEN
				WebserviceDownload.send := TRUE;
			// Sending data finished
			ELSIF (WebserviceDownload.send = TRUE) THEN
				WebserviceDownload.send := FALSE;
				rec_state := DAT_DOWNLOAD_4;
			// ----------------------------------------------------------------------------------------
			// Error
			ELSIF (WebserviceDownload.status <> ERR_FUB_BUSY AND WebserviceDownload.status <> OK) THEN
				rec_state := CreateError(ADR(RECORDER), WebserviceDownload.status, "error sending web response", rec_state);
			END_IF
		// --------------------------------------------------------------------------------------------------------------------
		// Download file - web service
		// --------------------------------------------------------------------------------------------------------------------
		DAT_DOWNLOAD_4:
			WebserviceDownload();

			// ----------------------------------------------------------------------------------------
			// Finish sending data
			IF (WebserviceDownload.phase = httpPHASE_WAITING) THEN
				RECORDER.VIS[RECORDER.PAR.VisuSlotID].DownloadFileUrl := '';
				WebserviceDownload.send := FALSE;
				RECORDER.CMD.Download	:= 0;
				rec_state := DAT_WAIT;
			// ----------------------------------------------------------------------------------------
			// Error
			ELSIF (WebserviceDownload.status <> ERR_FUB_BUSY) THEN
				rec_state := CreateError(ADR(RECORDER), WebserviceDownload.status, "error sending web response", rec_state);
			END_IF
		// --------------------------------------------------------------------------------------------------------------------
		// Load configuration
		// --------------------------------------------------------------------------------------------------------------------
		DAT_LOAD_VARS:
			// ----------------------------------------------------------------------------------------
			// Initialize file open structure
			FOpen.enable	:= TRUE;
			FOpen.pDevice 	:= ADR(DeviceName);
			FOpen.pFile		:= ADR(DAT_CONFIG);
			FOpen();

			// ----------------------------------------------------------------------------------------
			// OK
			IF (FOpen.status = OK) THEN
				// Make sure file fits into memory
				IF(FOpen.filelen <= DAT_DOWNLOAD_SIZE) THEN
					// Clear memory and reset web service
					brsmemset(AsMemPartAllocClear_0.mem, 0, DAT_DOWNLOAD_SIZE);
					rec_state := DAT_LOAD_VARS_1;
				// File is too large
				ELSE
					tmpWStr1 := "variable config file exceeds maximum buffer size of ";
					brsitoa(DAT_DOWNLOAD_SIZE, ADR(tmpStr1));
					brwcsconv(ADR(tmpWStr2),ADR(tmpStr1), brwU8toUC);
					brwcscat(ADR(tmpWStr1), ADR(tmpWStr2));
					brwcscat(ADR(tmpWStr1), ADR(" bytes"));
					rec_state := CreateError(ADR(RECORDER), ERR_MEM_DOWNLOAD, tmpWStr1, rec_state);
				END_IF;
			// ----------------------------------------------------------------------------------------
			// Error
			ELSIF (FOpen.status <> ERR_FUB_BUSY) THEN
				rec_state := CreateError(ADR(RECORDER), FOpen.status, "error opening variable config file", rec_state);
			END_IF
		// --------------------------------------------------------------------------------------------------------------------
		// Load configuration
		// --------------------------------------------------------------------------------------------------------------------
		DAT_LOAD_VARS_1:
			// ----------------------------------------------------------------------------------------
			// Initialize file read structure
			FRead.enable	:= TRUE;
			FRead.ident		:= FOpen.ident;
			FRead.len		:= FOpen.filelen;
			FRead.pDest		:= AsMemPartAllocClear_0.mem;
			FRead();

			// ----------------------------------------------------------------------------------------
			// OK
			IF (FRead.status = OK) THEN
				rec_state := DAT_LOAD_VARS_2;
			// ----------------------------------------------------------------------------------------
			// Error
			ELSIF (FRead.status <> ERR_FUB_BUSY) THEN
				rec_state := CreateError(ADR(RECORDER), FRead.status, "error reading variable config file", rec_state);
			END_IF
		// --------------------------------------------------------------------------------------------------------------------
		// Load configuration
		// --------------------------------------------------------------------------------------------------------------------
		DAT_LOAD_VARS_2:
			// ----------------------------------------------------------------------------------------
			// Initialize file close structure
			FClose.enable	:= TRUE;
			FClose.ident	:= FOpen.ident;
			FClose();

			// ----------------------------------------------------------------------------------------
			// OK
			IF (FClose.status = OK) THEN
				// Reset variable list
				brsmemset(ADR(DAT_VAR_LIST), 0, SIZEOF(DAT_VAR_LIST));
				ida := 0;
				idc := 1;
				rec_state := DAT_LOAD_VARS_3;
			// ----------------------------------------------------------------------------------------
			// Error
			ELSIF (FClose.status <> ERR_FUB_BUSY) THEN
				rec_state := CreateError(ADR(RECORDER), FClose.status, "error closing variable config file", rec_state);
			END_IF
		// --------------------------------------------------------------------------------------------------------------------
		// Load configuration
		// --------------------------------------------------------------------------------------------------------------------
		DAT_LOAD_VARS_3:
			idb := IsInstr(AsMemPartAllocClear_0.mem + ida, ADR(";"));
			IF idb > 0 THEN
				brsmemcpy(ADR(DAT_VAR_LIST[idc]), AsMemPartAllocClear_0.mem + ida, idb);
				ReplaceString(ADR(DAT_VAR_LIST[idc]), ADR('$n'), ADR(''), FALSE);
				ReplaceString(ADR(DAT_VAR_LIST[idc]), ADR('$r'), ADR(''), FALSE);
				ida := ida + idb + 1;

				IF ida >= FOpen.filelen THEN
					// Reset data structure and trigger name refresh for vis
					brsmemset(ADR(RECORDER.DAT), 0, SIZEOF(RECORDER.DAT));
					brsmemset(ADR(RecordNumOld), 16#FF, SIZEOF(RecordNumOld));
					pvCnt := 1;
					rec_state := DAT_CFG_READ;
				ELSE
					// Make sure we have enough slots for variables
					idc := idc + 1;
					IF idc > SIZEOF(DAT_VAR_LIST)/SIZEOF(DAT_VAR_LIST[1]) THEN
						rec_state := CreateError(ADR(RECORDER), ERR_DAT_VAR_NAME_NUM, "variable config file contains too many variables", rec_state);
					END_IF
				END_IF
			ELSE
				rec_state := CreateError(ADR(RECORDER), ERR_DAT_VAR_NAME_END, "variable config file contains too many variables", rec_state);
			END_IF
		// --------------------------------------------------------------------------------------------------------------------
		// Error
		// --------------------------------------------------------------------------------------------------------------------
		DAT_ERROR:
			RECORDER.StatusText := "error state triggered on web client ID ";
			tmpWStr1 := DINT_TO_WSTRING(RECORDER.PAR.VisuSlotID);
			brwcscat(ADR(RECORDER.StatusText), ADR(tmpWStr1));
			// --------------------------------------------------------------------------------------------------------------------
			// Make sure we dont exceed maximum number of web clients
			IF(RECORDER.PAR.VisuSlotID <= DAT_MAX_CLIENTS_ID) THEN
				RECORDER.VIS[RECORDER.PAR.VisuSlotID].ShowMessageBoxError := TRUE;
			END_IF
			// --------------------------------------------------------------------------------------------------------------------
			// Return to idle state
			IF RECORDER.CMD.ErrorReset THEN
				// Reset function blocks
				MpDataRecorder_0.Enable := FALSE;
				MpDataRecorder_0.Record := FALSE;
				MpDataRecorder_0.Trigger := FALSE;
				mappDataCfg.Enable := FALSE;
				mappDataCfg.Save := FALSE;
				mappDataCfg.Load := FALSE;

				FOR idx:=1 TO DAT_VAR_NUM DO
					MpRecorderRegPar_0[idx].Enable := FALSE;
					IF(DAT_VAR_LIST[idx] = '') THEN
						EXIT;
					END_IF
				END_FOR;

				// Reset error structure
				brsmemset(ADR(RECORDER.ERR), 0, SIZEOF(RECORDER.ERR));
				RECORDER.StatusText := "";
				RECORDER.CMD.ErrorReset := FALSE;
				RECORDER.VIS[RECORDER.PAR.VisuSlotID].ShowMessageBoxError := FALSE;
				rec_state := DAT_WAIT;
			END_IF;
			brsmemset(ADR(RECORDER.CMD), 0, SIZEOF(RECORDER.CMD));
	END_CASE

	// --------------------------------------------------------------------------------------------------------------------
	// Cyclic function calls
	FOR idx:=1 TO DAT_VAR_NUM DO
		MpRecorderRegPar_0[idx]();
		IF(DAT_VAR_LIST[idx] = '') THEN
			EXIT;
		END_IF
	END_FOR;
	MpDataRecorder_0.Enable := TRUE;
	MpDataRecorder_0.MpLink := ADR(MpComGetLink_0.MpLink);
	MpDataRecorder_0.DeviceName := ADR(DeviceName);
	MpDataRecorder_0();
	mappDataCfg.Enable := TRUE;
	mappDataCfg.MpLink := ADR(MpComGetLink_0.MpLink);
	mappDataCfg.Configuration := ADR(MpDataRecorderCfg);
	mappDataCfg();

END_PROGRAM
```

#### Exit.st
```iecst
PROGRAM _EXIT
	// --------------------------------------------------------------------------------------------------------------------
	// Cyclic function calls
	FOR idx:=1 TO DAT_VAR_NUM DO
		MpRecorderRegPar_0[idx](Enable := FALSE);
		IF(DAT_VAR_LIST[idx] = '') THEN
			EXIT;
		END_IF
	END_FOR;
	MpDataRecorder_0(Enable := FALSE);

END_PROGRAM
```

#### RecorderVariables.var - Local variables
```iecst
(*------------------------------------------------------------------------------------------------------------------------------------------------------------------------------------------------------------------------*)
(*Local constants*)
VAR CONSTANT
	OK : USINT := 0; (*Constant for status OK *)
END_VAR
(*------------------------------------------------------------------------------------------------------------------------------------------------------------------------------------------------------------------------*)
(*Local Variables*)
VAR
	RECORDER : REFERENCE TO datMAIN; (*Local recorder structure*)
	DeviceName : STRING[80]; (*Device name where the records are stored*)
	RecordName : STRING[DAT_NAME_LENGTH]; (*Local recorder name*)
	RecordFilterOld : ARRAY[0..DAT_MAX_CLIENTS_ID] OF WSTRING[DAT_NAME_LENGTH]; (*Track filter change *)
	RecordNumOld : ARRAY[0..DAT_MAX_CLIENTS_ID] OF UINT;
	rec_state : datSTATE := DAT_WAIT; (*Main step index *)
	animation : USINT := 0; (*Animation for working status	*)
	VisuSlotID : USINT; (*Slot of the visualization that is current used*)
	idx : UINT; (*Index*)
	idy : UINT; (*Index*)
	ida : UDINT; (*Index*)
	idb : UDINT; (*Index*)
	idc : UDINT; (*Index*)
	has_oversized_items : BOOL; (*Indicates that at least one recorder name exceeds the maximum length*)
	DownloadTimeout : TON_10ms; (*Timeout when download must finish*)
	ResponseHeader : httpResponseHeader_t; (*Response header for download*)
	ResponseHeaderData : STRING[300]; (*Response header data*)
	tmpStr1 : STRING[200]; (*Temporary string variable *)
	tmpWStr1 : WSTRING[DAT_VIS_LENGTH]; (*Temporary unicode string variable *)
	tmpWStr2 : WSTRING[DAT_VIS_LENGTH]; (*Temporary unicode string variable *)
	lDirReadData : fiDIR_READ_EX_DATA; (*File information structure*)
	taskID : UDINT; (*Task ID*)
	taskGroup : USINT; (*Task Group*)
	taskStatus : UINT; (*Status of task information*)
	pvADR : UDINT; (*Adress of global variable structure*)
	pvLEN : UDINT; (*Lenght of global variable structure*)
	pvStatus : UINT; (*Status of global variable information*)
	pvCnt : UINT; (*Counter for variable registration*)
	DoubleClickRecordName : ARRAY[0..DAT_MAX_CLIENTS_ID] OF TON_10ms; (*Timer for double click detection*)
	MpDataRecorderCfg : MpDataRecorderConfigType; (*Recorder configuration*)
END_VAR
(*------------------------------------------------------------------------------------------------------------------------------------------------------------------------------------------------------------------------*)
(*Local function calls*)
VAR
	DInfo : DirInfo;
	DOpen : DirOpen;
	DRead : DirReadEx;
	DClose : DirClose;
	FDelete : FileDelete;
	FOpen : FileOpen;
	FRead : FileReadEx;
	FClose : FileClose;
	MpDataRecorder_0 : MpDataRecorder;
	MpRecorderRegPar_0 : ARRAY[1..DAT_VAR_NUM] OF MpDataRegPar;
	mappDataCfg : MpDataRecorderConfig;
	MpComGetLink_0 : MpComGetLink;
	AsMemPartCreate_0 : AsMemPartCreate;
	AsMemPartAllocClear_0 : AsMemPartAllocClear;
	WebserviceDownload : httpService := (0);
END_VAR
(*------------------------------------------------------------------------------------------------------------------------------------------------------------------------------------------------------------------------*)
(*Error numbers*)
VAR CONSTANT
	ERR_MEM_ALLOC : UINT := 50400; (*Memory allocation for file upload and download failed*)
	ERR_MEM_DOWNLOAD : UINT := 50410; (*Size of download file exceeds maximum*)
	ERR_TIMEOUT_DOWNLOAD : UINT := 50420; (*Download response timed out*)
	ERR_DAT_TOO_MANY_CLIENTS : DINT := 50010; (*More than 3 clients try to connect to recorder management*)
	ERR_DAT_NAME_EMPTY : DINT := 50100; (*Recorder name is empty*)
	ERR_DAT_NAME_LENGTH : DINT := 50103; (*One or more recorder names exceeds maximum length*)
	ERR_DAT_DEV_NAME_EMPTY : DINT := 50110; (*Device name is empty*)
	ERR_DAT_VAR_NAME_EMPTY : DINT := 50120; (*Variable name is empty*)
	ERR_DAT_VAR_NAME_NUM : DINT := 50121; (*Config file contains too many variable names*)
	ERR_DAT_VAR_NAME_END : DINT := 50122; (*Cannot find end of varaible name in config file*)
	ERR_DAT_NOT_INITIALIZED : DINT := 50130; (*Recorder management is not initialized*)
	ERR_DAT_MPLINK : DINT := 50160; (*MpLink name is incorrect*)
	ERR_DAT_MAX_NUM : DINT := 50200; (*Maximum number of recorders reached*)
	ERR_DAT_TASK_NAME : DINT := 50300; (*Task name is incorrect*)
END_VAR
```

#### LocalFunctions.fun - Local function definition
```iecst
FUNCTION ReplaceString : BOOL
	VAR_INPUT
		dataSTR : UDINT;
		searchSTR : UDINT;
		replaceSTR : UDINT;
		first : BOOL;
	END_VAR
	VAR
		idx : UDINT;
	END_VAR
END_FUNCTION

FUNCTION CreateError : datSTATE
	VAR_INPUT
		RECORDER : REFERENCE TO datMAIN;
		No : DINT;
		Text : WSTRING[200];
		State : datSTATE;
	END_VAR
END_FUNCTION

FUNCTION CreateMessage : BOOL
	VAR_INPUT
		TargetString : UDINT;
		Text : UDINT;
		RecordName : UDINT;
		VisuSlotID : USINT;
	END_VAR
	VAR
		VisuSlotIDStr : WSTRING[5];
		tmpWStr1 : WSTRING[200];
	END_VAR
END_FUNCTION

FUNCTION InsertRecName : UINT
	VAR_INPUT
		RECORDER : REFERENCE TO datMAIN;
		new_name : STRING[DAT_NAME_LENGTH];
	END_VAR
	VAR
		idx : INT;
		idy : INT;
		lSort : DINT;
	END_VAR
END_FUNCTION

FUNCTION IsInstr : UDINT
	VAR_INPUT
		string1 : UDINT;
		string2 : UDINT;
	END_VAR
	VAR
		idx : UDINT;
	END_VAR
END_FUNCTION

FUNCTION WorkingStatus : USINT
	VAR_INPUT
		RECORDER : REFERENCE TO datMAIN;
		str : UDINT;
		animation : USINT;
	END_VAR
END_FUNCTION

FUNCTION String2DataProvider : BOOL
	VAR_INPUT
		SourceString : UDINT;
		TargetString : UDINT;
	END_VAR
END_FUNCTION
```

#### LocalFunctions.st - Local function code
```iecst
//******************************************************************************************************
// Create mappView data provider string
//******************************************************************************************************
FUNCTION String2DataProvider
	brsstrcpy(TargetString, ADR('{"value":"'));
	brsstrcat(TargetString, SourceString);
	brsstrcat(TargetString, ADR('","text":"'));
	brsstrcat(TargetString, SourceString);
	brsstrcat(TargetString, ADR('"}'));

	String2DataProvider := TRUE;
END_FUNCTION

//******************************************************************************************************
// Create error
//******************************************************************************************************
FUNCTION CreateError
	RECORDER.StatusNo := No;
	RECORDER.ERR.State := State;
	RECORDER.ERR.Text := Text;
	CreateError := DAT_ERROR;
END_FUNCTION

//******************************************************************************************************
// Create status meesage
//******************************************************************************************************
FUNCTION CreateMessage
	brwcscpy(ADR(tmpWStr1), Text);
	brwcscat(ADR(tmpWStr1), ADR(" "));
	brwcscat(ADR(tmpWStr1), RecordName);
	brwcscat(ADR(tmpWStr1), ADR(" on web client ID "));
	VisuSlotIDStr := DINT_TO_WSTRING(VisuSlotID);
	brwcscat(ADR(tmpWStr1), ADR(VisuSlotIDStr));
	brwcscpy(TargetString, ADR(tmpWStr1));

	CreateMessage := TRUE;
END_FUNCTION

//******************************************************************************************************
// Working status
//******************************************************************************************************
FUNCTION WorkingStatus
	animation := animation+1;

	IF (animation = 80) THEN
		animation := 0;
	END_IF

	brsmemset(ADR(RECORDER.StatusText), 0, SIZEOF(RECORDER.StatusText));
	brwcscpy(ADR(RECORDER.StatusText), str);
	CASE(animation) OF
		0..19	: brwcscat(ADR(RECORDER.StatusText), ADR("/"));
		20..39	: brwcscat(ADR(RECORDER.StatusText), ADR("-"));
		40..59	: brwcscat(ADR(RECORDER.StatusText), ADR("\"));
		60..79	: brwcscat(ADR(RECORDER.StatusText), ADR("|"));
	END_CASE;
	WorkingStatus := animation;
END_FUNCTION

//******************************************************************************************************
// Fill new folder or directory name
//******************************************************************************************************
FUNCTION InsertRecName
	// Set up start values for iteration
	IF (RECORDER.DAT.RecordNum <> 0) THEN
		idy := RECORDER.DAT.RecordNum - 1;
	END_IF
	idx := idy;

	// Start iteration	search
	WHILE (idy > 1) DO
		// Check current entry
		lSort := brsstrcmp(ADR(new_name), ADR(RECORDER.DAT.RecordNames[idy]));
		// Solve new search range
		IF (idy MOD 2 = 0) THEN
			idy := idy / 2;
		ELSE
			idy := idy / 2 + 1;
		END_IF
		// New range is lower or higher than current
		IF (lSort > 0) THEN
			idx := idx + idy;
			IF (idx > UINT_TO_INT(RECORDER.DAT.RecordNum)) THEN
				idx := RECORDER.DAT.RecordNum;
			END_IF
		ELSE
			idx := idx - idy;
			IF (idx < 1) THEN
				idx := 1;
			END_IF
		END_IF
	END_WHILE;

	// New entry is this, next or previous
	lSort := brsstrcmp(ADR(new_name), ADR(RECORDER.DAT.RecordNames[idx]));
	IF (lSort > 0 AND idx <> UINT_TO_INT(RECORDER.DAT.RecordNum)) THEN
		idx := idx +1;
	ELSIF (idx > 0) THEN
		lSort := brsstrcmp(ADR(new_name), ADR(RECORDER.DAT.RecordNames[idx-1]));
		IF (lSort < 0) THEN
			idx := idx - 1;
		END_IF
	END_IF

	// Move all data entrys backwards and fill in new entry
	IF(idx < DAT_MAX_NUM) THEN
		brsmemmove(ADR(RECORDER.DAT.RecordNames[idx+1]),ADR(RECORDER.DAT.RecordNames[idx]), (RECORDER.DAT.RecordNum - idx) * SIZEOF(RECORDER.DAT.RecordNames[1]));
	END_IF
	brsstrcpy(ADR(RECORDER.DAT.RecordNames[idx]), ADR(new_name));

	RECORDER.DAT.RecordNum := RECORDER.DAT.RecordNum + 1;
	InsertRecName := idx;
END_FUNCTION

//******************************************************************************************************
// Is second string in first string
//******************************************************************************************************
FUNCTION IsInstr
	IF (brsstrlen(string1) >= brsstrlen(string2)) THEN
		FOR idx:=0 TO brsstrlen(string1) - brsstrlen(string2) DO
			IF (brsmemcmp(string1 + idx, string2, brsstrlen(string2)) = 0) THEN
				IsInstr := idx;
				EXIT;
			END_IF
		END_FOR;
	END_IF
END_FUNCTION

//******************************************************************************************************
// Find and replace string
//******************************************************************************************************
FUNCTION ReplaceString
	IF (brsstrlen(dataSTR) >= brsstrlen(searchSTR)) THEN
		FOR idx:=0 TO brsstrlen(dataSTR) - brsstrlen(searchSTR) DO
			IF (brsmemcmp(dataSTR + idx, searchSTR, brsstrlen(searchSTR)) = 0) THEN
				// Move data around
				brsmemmove(dataSTR + idx + brsstrlen(replaceSTR), dataSTR + idx + brsstrlen(searchSTR), brsstrlen(dataSTR) - brsstrlen(searchSTR) + 1);
				brsmemcpy(dataSTR + idx, replaceSTR, brsstrlen(replaceSTR));
				// Set found flag and exit if only one hit is needed
				ReplaceString := TRUE;
				IF(first) THEN
					EXIT;
				END_IF
				// Correct index for next search
				IF(brsstrlen(replaceSTR) > 0) THEN
					idx := idx + brsstrlen(replaceSTR);
				END_IF
				idx := idx - 1;
				// Exit if no data is left
				IF (brsstrlen(dataSTR) = 0 OR brsstrlen(dataSTR) < brsstrlen(searchSTR)) THEN
					EXIT;
				END_IF
			END_IF
		END_FOR;
	END_IF
END_FUNCTION
```

### Program Logical/mappRecorder/YourTask (IEC)

#### YourVariables.var
```iecst
VAR
	Position : REAL;
	MotorSpeed : DINT;
	Temperature2 : DINT;
	Temperature1 : DINT;
END_VAR
```

#### Main.st
```iecst
// --------------------------------------------------------------------------------------------------------------------
// Use this task to add your own code for recorder managment
// --------------------------------------------------------------------------------------------------------------------
PROGRAM _INIT
	// Sample record data, the global array DAT_VAR_LIST define what variables belong to a record
	Temperature1 := 123;
	Temperature2 := 130;
	MotorSpeed := 1000;
	Position := 0;
	Recorder_1;
END_PROGRAM

PROGRAM _CYCLIC
	(* Insert code here *)

END_PROGRAM

PROGRAM _EXIT
	(* Insert code here *)

END_PROGRAM
```

### changelog.txt
```
Version 0.6 (05.05.2023)
- Updated Automation Studio and mapp components
- Added new command LoadConfig to load a variable list from a file
- Minor bug fixes

Version 0.5 (05.02.2021)
- Fixed memory violation when file exceeds download buffer size

Version 0.4 (15.06.2020)
- Only start recording when FUB is active
- Changed some parameters to constants
- Simplified configuration
- Added more error messages
- Added the possibility to define multiple variables
- Moved status text to main structure
- Moved error no up to main structure and renamed it to StatusNo
- Rercord name can now be defined at RecordNameNew

Version 0.3
- Fixed oversized item flag is not reset
- Fixed ReplaceString function call
- Update mapp to version 5.8.1

Version 0.2
- Fixed download not working when downloading the same file again

Version 0.1
- First public release
```

- var_list.csv (not shown)

### Types.typ - not listed in the package file held
```iecst
(*------------------------------------------------------------------------------------------------------------------------------------------------------------------------------------------------------------------------*)
(*Global enumerations*)

TYPE
	datSTATE :
		( (*Recorder managment state machine*)
		DAT_WAIT,
		DAT_REG_VAR,
		DAT_READ_DIR,
		DAT_READ_DIR_1,
		DAT_READ_DIR_2,
		DAT_READ_DIR_3,
		DAT_RECORD,
		DAT_DELETE,
		DAT_VIEW,
		DAT_DOWNLOAD,
		DAT_DOWNLOAD_1,
		DAT_DOWNLOAD_2,
		DAT_DOWNLOAD_3,
		DAT_DOWNLOAD_4,
		DAT_ERROR
		);
END_TYPE

(*------------------------------------------------------------------------------------------------------------------------------------------------------------------------------------------------------------------------*)
(*Global structure*)

TYPE
	datERR : 	STRUCT  (*Recorder managment error structure*)
		Text : WSTRING[200]; (* Error text *)
		No : DINT; (* Error number *)
		State : datSTATE; (* Error step *)
	END_STRUCT;
	datCMD : 	STRUCT  (*Recorder managment command structure*)
		Init : BOOL := TRUE; (*Initialize recorder structure*)
		Record : BOOL; (*Enable recording*)
		Trigger : BOOL; (*Trigger recording*)
		Delete : BOOL; (*Delete selected file *)
		View : BOOL; (*View selected file*)
		Download : BOOL; (*Download selected file*)
		ErrorReset : BOOL; (*Reset pending errors*)
	END_STRUCT;
	datPAR : 	STRUCT  (*Recorder managment parameter structure*)
		RecordVariable : STRING[200]; (*Name of the variable where the data is stored*)
		RecordName : STRING[200]; (*Record name for command delete and view*)
		RecordMode : MpDataRecordModeEnum; (*Recording mode*)
		RecordInterval : TIME := T#2000ms;
		IsRecording : BOOL; (*Indicates that recording is active*)
		SamplesNum : UDINT; (*Number of recorded samples*)
		DeviceName : STRING[100]; (*Device name where the records are stored*)
		MpLink : MpComIdentType; (*MpLink from mappRecorder*)
		Initialized : BOOL; (*Indicates that recorder managment was initialized*)
		VisuSlotID : USINT; (*ID for connected web connection*)
	END_STRUCT;
	datDAT : 	STRUCT  (*Recorder managment data structure*)
		RecordNames : ARRAY[0..DAT_MAX_NUM]OF STRING[DAT_NAME_LENGTH]; (*Recorder unicode name*)
		RecordNum : UINT; (*Number of recorded files*)
		Status : WSTRING[100]; (*Shows the result of the last command*)
	END_STRUCT;
	datVIS : 	STRUCT  (*Recorder managment visualization structure*)
		RecordNames : ARRAY[0..DAT_MAX_NUM]OF STRING[DAT_VIS_LENGTH]; (*Recorder file size*)
		RecordNum : UINT; (*Number of records*)
		RecordFilter : STRING[DAT_NAME_LENGTH]; (*Filter for record names*)
		RecordSelected : STRING[DAT_VIS_LENGTH]; (*Selected record for command delete or view*)
		RecordDoubleClick : USINT; (*TrackDoubleClick event*)
		EnableButtons : BOOL;
		ViewFilePath : STRING[DAT_VIS_LENGTH]; (*Full path for viewing file*)
		ViewFile : BOOL; (*Show message box on error*)
		DownloadFileUrl : STRING[200]; (*File upload and download url*)
		ShowMessageBoxError : BOOL; (*Show message box on error*)
	END_STRUCT;
	datMAIN : 	STRUCT  (*Recorder managment main structure*)
		CMD : datCMD; (* Command structure *)
		PAR : datPAR; (* Parameter structure *)
		DAT : datDAT; (*Data structure*)
		VIS : ARRAY[0..DAT_MAX_CLIENTS_ID]OF datVIS; (*Visualization structure*)
		ERR : datERR; (* Error structure *)
	END_STRUCT;
END_TYPE

(*------------------------------------------------------------------------------------------------------------------------------------------------------------------------------------------------------------------------*)
(*Structure that contains the recorder variables*)

TYPE
	datVariable : 	STRUCT
		Temperature1 : INT := 11;
		Temperature2 : INT := 22;
		MotorSpeed : DINT := 33;
		Position : REAL := 44.55;
	END_STRUCT;
END_TYPE
```

### Variables.var - not listed in the package file held
```iecst
(*------------------------------------------------------------------------------------------------------------------------------------------------------------------------------------------------------------------------*)
(*Configuration for recorder managment*)
VAR CONSTANT
	DAT_MAX_NUM : USINT := 100; (*Maximum number of record files*)
	DAT_NAME_LENGTH : USINT := 40; (*Maximum length for a record name*)
	DAT_VIS_LENGTH : USINT := 120; (*Make this DAT_NAME_LENGTH  x3*)
	DAT_MAX_CLIENTS_ID : USINT := 2; (*Highest client ID for concurrent web client connections. Do not change this number.*)
END_VAR
VAR
	DAT_VIEW_FILTER : ARRAY[0..9] OF STRING[5] := ['csv','xml',8('')]; (*Files extensions than can be used with the view command*)
END_VAR
VAR CONSTANT
	DAT_DOWNLOAD_SIZE : UDINT := 500000; (*Maximum size of memory allocated for uploading and downloading files*)
END_VAR
VAR
	Recorder_1 : datMAIN; (*Global record structure. The name must match the task name of the recorder managment.*)
	RecorderData : datVariable; (*Structure that contains the recorder variables*)
END_VAR
```

Listed in the project but not available here: Logical/Global.typ, Logical/Global.var
